            "740338" : Bool;   // (WRN) UNIT 1 STATION 04 SAFETY DOOR UNLOCK WITH CYCLE RUNNING REQUESTED
            "740341" : Bool;   // (WRN) UNIT 2 MAIN SAFETY DOOR UNLOCK WITH CYCLE RUNNING REQUESTED
            "740342" : Bool;   // (WRN) UNIT 2 STATION 02 SAFETY DOOR UNLOCK WITH CYCLE RUNNING REQUESTED
            "740343" : Bool;   // (WRN) UNIT 2 STATION 04 SAFETY DOOR UNLOCK WITH CYCLE RUNNING REQUESTED
            "740350" : Bool;   // (WRN) SAFETY DOOR BYPASS NOT SELECTED
            "740351" : Bool;   // (WRN) ANY SAFETY DOOR NOT CLOSED AND LOCKED
            "740361" : Bool;   // (WRN) UNIT 1 POWDER FEEDER DISABLED
            "740362" : Bool;   // (WRN) UNIT 1 PYROMETER DISABLED
            "740363" : Bool;   // (WRN) UNIT 1 LASER DISABLED
            "740364" : Bool;   // (WRN) UNIT 1 STATION 3 MEASURING PC DISABLED
            "740365" : Bool;   // (WRN) UNIT 1 STATION 3 COAXIAL PC DISABLED
            "740366" : Bool;   // (WRN) UNIT 1 FIXTURE 1 & 4 DISABLED
            "740367" : Bool;   // (WRN) UNIT 1 FIXTURE 2 & 3 DISABLED
            "740371" : Bool;   // (WRN) UNIT 2 POWDER FEEDER DISABLED
            "740372" : Bool;   // (WRN) UNIT 2 PYROMETER DISABLED
            "740373" : Bool;   // (WRN) UNIT 2 LASER DISABLED
            "740374" : Bool;   // (WRN) UNIT 2 STATION 2 MEASURING PC DISABLED
            "740375" : Bool;   // (WRN) UNIT 2 STATION 3 MEASURING PC DISABLED
            "740376" : Bool;   // (WRN) UNIT 2 STATION 3 COAXIAL PC DISABLED
            "740377" : Bool;   // (WRN) UNIT 2 FIXTURE 1 & 4 DISABLED
            "740378" : Bool;   // (WRN) UNIT 2 FIXTURE 2 & 3 DISABLED
            "740380" : Bool;   // (WRN) UNIT 03 MEASURING PC A DISABLED
            "740381" : Bool;   // (WRN) UNIT 03 MEASURING PC B DISABLED
            "740390" : Bool;   // (WRN) HOLA PC DISABLED
            "740440" : Bool;   // (WRN) QUALITY PART INSPECTION AFTER PART COUNT REACHED
            "740456" : Bool;   // (WRN) QUALITY PART INSPECTION AFTER PART TYPE CHANGE
            "740472" : Bool;   // (WRN) QUALITY PART INSPECTION AFTER FIRST CYCLE
            "740600" : Bool;   // (WRN) C11 HIGH TEMPERATURE PREALARM
            "740601" : Bool;   // (WRN) C12 HIGH TEMPERATURE PREALARM
            "740602" : Bool;   // (WRN) C13 HIGH TEMPERATURE PREALARM
            "740603" : Bool;   // (WRN) C14 HIGH TEMPERATURE PREALARM
            "740608" : Bool;   // (WRN) C21 HIGH TEMPERATURE PREALARM
            "740610" : Bool;   // (WRN) C23 HIGH TEMPERATURE PREALARM
            "740611" : Bool;   // (WRN) C24 HIGH TEMPERATURE PREALARM
            "741000" : Bool;   // (WRN) UNIT 1 ASPIRATION SYSTEM PRESSURE TOO LOW WARNING
            "741001" : Bool;   // (WRN) UNIT 1 ASPIRATION SYSTEM PRESSURE TOO HIGH WARNING
            "741002" : Bool;   // (WRN) UNIT 2 ASPIRATION SYSTEM PRESSURE TOO LOW WARNING
            "741003" : Bool;   // (WRN) UNIT 2 ASPIRATION SYSTEM PRESSURE TOO HIGH WARNING
            "741240" : Bool;   // (WRN) MACHINE COOLING SYSTEM INPUT SENSOR FLOW LOW
            "741241" : Bool;   // (WRN) MACHINE COOLING SYSTEM INPUT SENSOR FLOW HIGH
            "741242" : Bool;   // (WRN) MACHINE COOLING SYSTEM INPUT SENSOR TEMPERATURE LOW
            "741243" : Bool;   // (WRN) MACHINE COOLING SYSTEM INPUT SENSOR TEMPERATURE HIGH
            "741245" : Bool;   // (WRN) MACHINE COOLING SYSTEM OUTPUT SENSOR FLOW LOW
            "741246" : Bool;   // (WRN) MACHINE COOLING SYSTEM OUTPUT SENSOR FLOW HIGH
            "741247" : Bool;   // (WRN) MACHINE COOLING SYSTEM OUTPUT SENSOR TEMPERATURE LOW
            "741248" : Bool;   // (WRN) MACHINE COOLING SYSTEM OUTPUT SENSOR TEMPERATURE HIGH
            "741256" : Bool;   // (WRN) UNIT 1 SHIELD AUXILIARY COOLING SYSTEM FLOW HIGH
            "741257" : Bool;   // (WRN) UNIT 1 SHIELD AUXILIARY COOLING SYSTEM FLOW LOW
            "741258" : Bool;   // (WRN) UNIT 1 SHIELD AUXILIARY COOLING SYSTEM TEMPERATURE HIGH
            "741259" : Bool;   // (WRN) UNIT 1 SHIELD AUXILIARY COOLING SYSTEM TEMPERATURE LOW
            "741264" : Bool;   // (WRN) UNIT 2 SHIELD AUXILIARY COOLING SYSTEM FLOW HIGH
            "741265" : Bool;   // (WRN) UNIT 2 SHIELD AUXILIARY COOLING SYSTEM FLOW LOW
            "741266" : Bool;   // (WRN) UNIT 2 SHIELD AUXILIARY COOLING SYSTEM TEMPERATURE HIGH
            "741267" : Bool;   // (WRN) UNIT 2 SHIELD AUXILIARY COOLING SYSTEM TEMPERATURE LOW
            "741272" : Bool;   // (WRN) UNIT 1 COOLING BUFFER AUXILIARY COOLING SYSTEM FLOW HIGH
            "741273" : Bool;   // (WRN) UNIT 1 COOLING BUFFER AUXILIARY COOLING SYSTEM FLOW LOW
            "741274" : Bool;   // (WRN) UNIT 1 COOLING BUFFER AUXILIARY COOLING SYSTEM TEMPERATURE HIGH
            "741275" : Bool;   // (WRN) UNIT 1 COOLING BUFFER AUXILIARY COOLING SYSTEM TEMPERATURE LOW
            "741280" : Bool;   // (WRN) UNIT 2 COOLING BUFFER AUXILIARY COOLING SYSTEM FLOW HIGH
            "741281" : Bool;   // (WRN) UNIT 2 COOLING BUFFER AUXILIARY COOLING SYSTEM FLOW LOW
            "741282" : Bool;   // (WRN) UNIT 2 COOLING BUFFER AUXILIARY COOLING SYSTEM TEMPERATURE HIGH
            "741283" : Bool;   // (WRN) UNIT 2 COOLING BUFFER AUXILIARY COOLING SYSTEM TEMPERATURE LOW
            "741400" : Bool;   // (WRN) LASER COOLING SYSTEM SENSOR INPUT U01 FLOW LOW
            "741401" : Bool;   // (WRN) LASER COOLING SYSTEM SENSOR INPUT U01 FLOW HIGH
            "741402" : Bool;   // (WRN) LASER COOLING SYSTEM SENSOR INPUT U01 TEMPERATURE LOW
            "741403" : Bool;   // (WRN) LASER COOLING SYSTEM SENSOR INPUT U01 TEMPERATURE HIGH
            "741405" : Bool;   // (WRN) LASER COOLING SYSTEM SENSOR 1 U01 FLOW LOW
            "741406" : Bool;   // (WRN) LASER COOLING SYSTEM SENSOR 1 U01 FLOW HIGH
            "741407" : Bool;   // (WRN) LASER COOLING SYSTEM SENSOR 1 U01 TEMPERATURE LOW
            "741408" : Bool;   // (WRN) LASER COOLING SYSTEM SENSOR 1 U01 TEMPERATURE HIGH
            "741410" : Bool;   // (WRN) LASER COOLING SYSTEM SENSOR 2 U01 FLOW LOW
            "741411" : Bool;   // (WRN) LASER COOLING SYSTEM SENSOR 2 U01 FLOW HIGH
            "741412" : Bool;   // (WRN) LASER COOLING SYSTEM SENSOR 2 U01 TEMPERATURE LOW
            "741413" : Bool;   // (WRN) LASER COOLING SYSTEM SENSOR 2 U01 TEMPERATURE HIGH
            "741415" : Bool;   // (WRN) LASER SYSTEM PROTECTION GAS U01 FLOW LOW
            "741416" : Bool;   // (WRN) LASER SYSTEM PROTECTION GAS U01 FLOW HIGH
            "741417" : Bool;   // (WRN) LASER SYSTEM PROTECTION GAS U01 TEMPERATURE LOW
            "741418" : Bool;   // (WRN) LASER SYSTEM PROTECTION GAS U01 TEMPERATURE HIGH
            "741440" : Bool;   // (WRN) LASER COOLING SYSTEM SENSOR INPUT U02 FLOW LOW
            "741441" : Bool;   // (WRN) LASER COOLING SYSTEM SENSOR INPUT U02 FLOW HIGH
            "741442" : Bool;   // (WRN) LASER COOLING SYSTEM SENSOR INPUT U02 TEMPERATURE LOW
            "741443" : Bool;   // (WRN) LASER COOLING SYSTEM SENSOR INPUT U02 TEMPERATURE HIGH
            "741445" : Bool;   // (WRN) LASER COOLING SYSTEM SENSOR 1 U02 FLOW LOW
            "741446" : Bool;   // (WRN) LASER COOLING SYSTEM SENSOR 1 U02 FLOW HIGH
            "741447" : Bool;   // (WRN) LASER COOLING SYSTEM SENSOR 1 U02 TEMPERATURE LOW
            "741448" : Bool;   // (WRN) LASER COOLING SYSTEM SENSOR 1 U02 TEMPERATURE HIGH
            "741450" : Bool;   // (WRN) LASER COOLING SYSTEM SENSOR 2 U02 FLOW LOW
            "741451" : Bool;   // (WRN) LASER COOLING SYSTEM SENSOR 2 U02 FLOW HIGH
            "741452" : Bool;   // (WRN) LASER COOLING SYSTEM SENSOR 2 U02 TEMPERATURE LOW
            "741453" : Bool;   // (WRN) LASER COOLING SYSTEM SENSOR 2 U02 TEMPERATURE HIGH
            "741455" : Bool;   // (WRN) LASER SYSTEM PROTECTION GAS U02 FLOW LOW
            "741456" : Bool;   // (WRN) LASER SYSTEM PROTECTION GAS U02 FLOW HIGH
            "741457" : Bool;   // (WRN) LASER SYSTEM PROTECTION GAS U02 TEMPERATURE LOW
            "741458" : Bool;   // (WRN) LASER SYSTEM PROTECTION GAS U02 TEMPERATURE HIGH
            "742040" : Bool;   // (WRN) UNIT 1 MACHINE NO PART AT FEED
            "742041" : Bool;   // (WRN) UNIT 2 MACHINE NO PART AT FEED
            "742043" : Bool;   // (WRN) UNIT 1 MACHINE DELIVERY OCCUPIED
            "742044" : Bool;   // (WRN) UNIT 2 MACHINE DELIVERY OCCUPIED
            "742120" : Bool;   // (WRN) UNIT 1 STATION 3 MEASURING COMPUTER WARNING: PLC-PC MINOR VERSIONS MISMATCH
            "742121" : Bool;   // (WRN) UNIT 1 STATION 3 CAMERA COMPUTER WARNING: PLC-PC MINOR VERSIONS MISMATCH
            "742122" : Bool;   // (WRN) UNIT 1 STATION 3 CAMERA COMPUTER WARNING: NO CAMERA AVAILABLE
            "742123" : Bool;   // (WRN) UNIT 1 STATION 3 CAMERA COMPUTER WARNING: MISSING LASER CALIBRATION
            "742124" : Bool;   // (WRN) UNIT 1 STATION 3 CAMERA COMPUTER WARNING: MISSING NOZZLE CALIBRATION
            "742128" : Bool;   // (WRN) UNIT 2 STATION 2 MEASURING COMPUTER WARNING: PLC-PC MINOR VERSIONS MISMATCH
            "742129" : Bool;   // (WRN) UNIT 2 STATION 3 MEASURING COMPUTER WARNING: PLC-PC MINOR VERSIONS MISMATCH
            "742130" : Bool;   // (WRN) UNIT 2 STATION 3 CAMERA COMPUTER WARNING: PLC-PC MINOR VERSIONS MISMATCH
            "742131" : Bool;   // (WRN) UNIT 2 STATION 3 CAMERA COMPUTER WARNING: NO CAMERA AVAILABLE
            "742132" : Bool;   // (WRN) UNIT 2 STATION 3 CAMERA COMPUTER WARNING: MISSING LASER CALIBRATION
            "742133" : Bool;   // (WRN) UNIT 2 STATION 3 CAMERA COMPUTER WARNING: MISSING NOZZLE CALIBRATION
            "742136" : Bool;   // (WRN) UNIT 3 FACE R MEASURING COMPUTER WARNING: PLC-PC MINOR VERSIONS MISMATCH
            "742137" : Bool;   // (WRN) UNIT 3 FACE N MEASURING COMPUTER WARNING: PLC-PC MINOR VERSIONS MISMATCH
            "742140" : Bool;   // (WRN) UNIT 1 PYROMETER PROCESS TEMPERATURE LOW
            "742141" : Bool;   // (WRN) UNIT 1 PYROMETER PROCESS TEMPERATURE HIGH
            "742142" : Bool;   // (WRN) UNIT 1 PYROMETER HEAD TEMPERATURE LOW
            "742143" : Bool;   // (WRN) UNIT 1 PYTOMETER HEAD TEMPERATURE HIGH
            "742144" : Bool;   // (WRN) UNIT 1 PYROMETER EMISSIVITY LOW
            "742145" : Bool;   // (WRN) UNIT 1 PYROMETER EMISSIVITY HIGH
            "742148" : Bool;   // (WRN) UNIT 2 PYROMETER PROCESS TEMPERATURE LOW
            "742149" : Bool;   // (WRN) UNIT 2 PYROMETER PROCESS TEMPERATURE HIGH
            "742150" : Bool;   // (WRN) UNIT 2 PYROMETER HEAD TEMPERATURE LOW
            "742151" : Bool;   // (WRN) UNIT 2 PYTOMETER HEAD TEMPERATURE HIGH
            "742152" : Bool;   // (WRN) UNIT 2 PYROMETER EMISSIVITY LOW
            "742153" : Bool;   // (WRN) UNIT 2 PYROMETER EMISSIVITY HIGH
            "743680" : Bool;   // TRADES CALL SPARE
            "743681" : Bool;   // TRADES CALL SPARE
            "743682" : Bool;   // TRADES CALL SPARE
            "743683" : Bool;   // TRADES CALL SPARE
            "743684" : Bool;   // TRADES CALL SPARE
            "743685" : Bool;   // TRADES CALL SPARE
            "743686" : Bool;   // TRADES CALL SPARE
            "743687" : Bool;   // TRADES CALL SPARE
         END_STRUCT;
         VERSIONS : Struct   // VERSIONS
            MINOR : Int := 31;
            MAJOR : Int := 1;
         END_STRUCT;
      END_STRUCT;
   END_VAR
BEGIN
END_DATA_BLOCK
